% RSLogix 500 project WN16_175300_PPWEXT_04_2.rss, saved by version 9.00.00.04 %
PROJECT "EDIRX88"    % processor: SLC 500, 1747-L541 %

PROGRAM FILES
  LAD 2   13 rungs
  LAD 3   63 rungs
  LAD 4   5 rungs
  LAD 5   96 rungs
  LAD 6   14 rungs
  LAD 7   7 rungs
  LAD 8   17 rungs
  LAD 9   51 rungs
  LAD 10   4 rungs
  LAD 11   3 rungs
  LAD 12   6 rungs
  LAD 13   6 rungs
  LAD 14   6 rungs
  LAD 15   14 rungs
  LAD 16   7 rungs
  LAD 17   12 rungs
  LAD 18   4 rungs
  LAD 19   3 rungs
  LAD 21   27 rungs
  LAD 22   4 rungs
  LAD 23   7 rungs
  LAD 24   36 rungs

DATA FILES
  O0 OUTPUT  7 elements
  I1 INPUT  11 elements
  S2 STATUS  164 elements
  B3 BINARY  51 elements
  T4 TIMER  34 elements
  C5 COUNTER  1 elements
  R6 CONTROL  1 elements
  N7 INTEGER  241 elements
  F8 FLOAT  1 elements
  N9   24 elements
  N10   19 elements
  B13   10 elements
  T14   21 elements
  N17   100 elements
  N19   24 elements
  N20   11 elements
  N30   30 elements
  T31   10 elements

LADDER 2
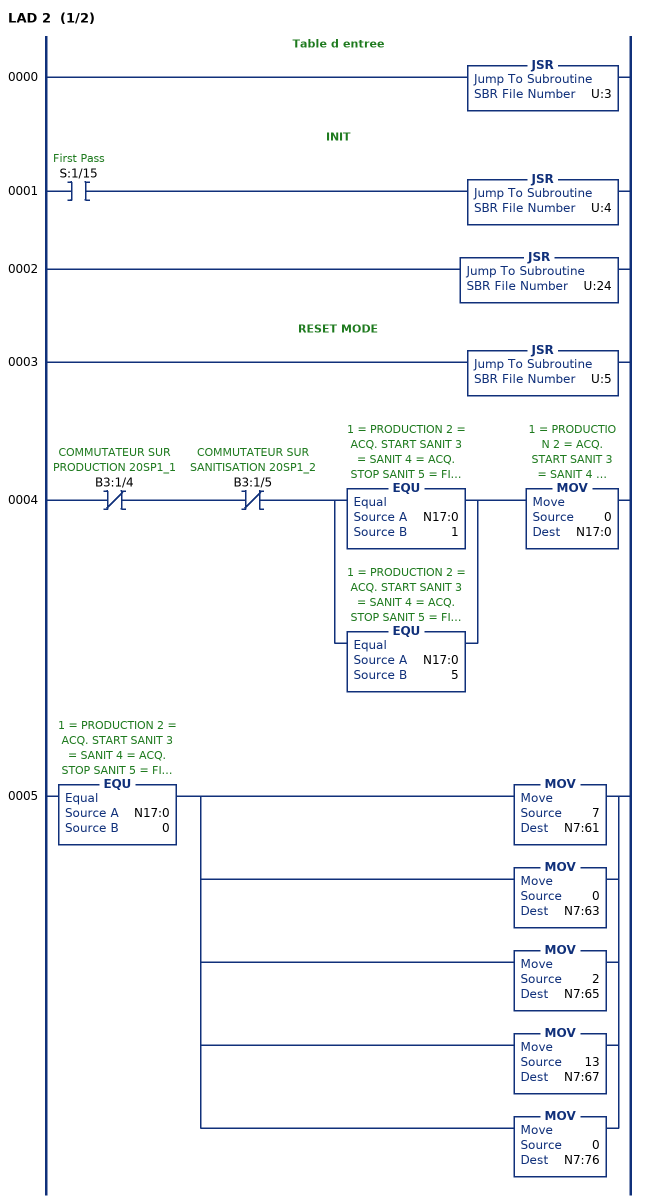
% Rung: 0 %
% TITLE: Table d entree %
SOR JSR U:3 EOR
% Rung: 1 %
% TITLE: INIT %
SOR XIC S:1/15 JSR U:4 EOR
%   S:1/15  "First Pass" %
% Rung: 2 %
SOR JSR U:24 EOR
% Rung: 3 %
% TITLE: RESET MODE %
SOR JSR U:5 EOR
% Rung: 4 %
SOR XIO B3:1/4 XIO B3:1/5 BST EQU N17:0 1 NXB EQU N17:0 5 BND MOV 0 N17:0 EOR
%   B3:1/4  20SP1_1  "COMMUTATEUR SUR PRODUCTION" %
%   B3:1/5  20SP1_2  "COMMUTATEUR SUR SANITISATION" %
%   N17:0  MODE  "1 = PRODUCTION 2 = ACQ. START SANIT 3 = SANIT 4 = ACQ. STOP SANIT 5 = FIN DE SANIT" %
% Rung: 5 %
SOR EQU N17:0 0 BST MOV 7 N7:61 NXB MOV 0 N7:63 NXB MOV 2 N7:65 NXB MOV 13 N7:67 NXB MOV 0 N7:76 BND EOR
%   N17:0  MODE  "1 = PRODUCTION 2 = ACQ. START SANIT 3 = SANIT 4 = ACQ. STOP SANIT 5 = FIN DE SANIT" %

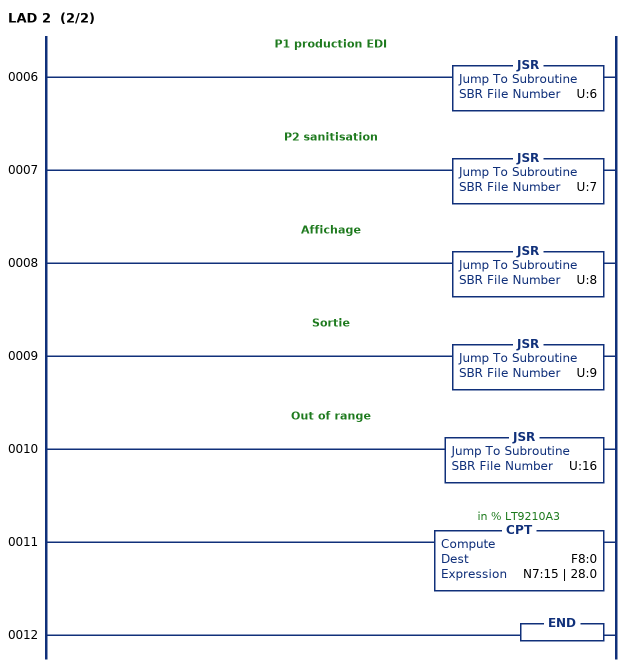
% Rung: 6 %
% TITLE: P1 production EDI %
SOR JSR U:6 EOR
% Rung: 7 %
% TITLE: P2 sanitisation %
SOR JSR U:7 EOR
% Rung: 8 %
% TITLE: Affichage %
SOR JSR U:8 EOR
% Rung: 9 %
% TITLE: Sortie %
SOR JSR U:9 EOR
% Rung: 10 %
% TITLE: Out of range %
SOR JSR U:16 EOR
% Rung: 11 %
SOR CPT F8:0 " N7:15 | 28.0 " EOR
%   F8:0  LT9210A3  "in %" %
%   N7:15  LT_VS_9210_A3 %
% Rung: 12 %
SOR END EOR

LADDER 3
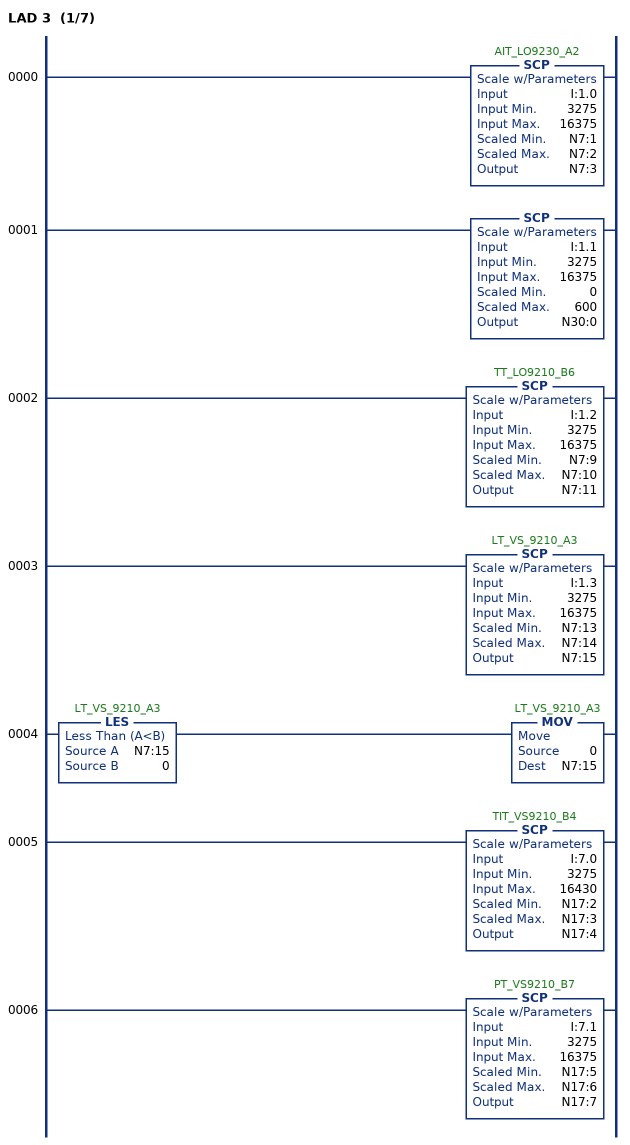
% Rung: 0 %
SOR SCP I:1.0 3275 16375 N7:1 N7:2 N7:3 EOR
%   N7:1  ZÉRO_AIT_LO9230_A2 %
%   N7:2  SPAN_AIT_LO9230_A2 %
%   N7:3  AIT_LO9230_A2 %
% Rung: 1 %
SOR SCP I:1.1 3275 16375 0 600 N30:0 EOR
% Rung: 2 %
SOR SCP I:1.2 3275 16375 N7:9 N7:10 N7:11 EOR
%   N7:9  ZÉRO_TT_LO9210_B6 %
%   N7:10  SPAN_TT_LO9210_B6 %
%   N7:11  TT_LO9210_B6 %
% Rung: 3 %
SOR SCP I:1.3 3275 16375 N7:13 N7:14 N7:15 EOR
%   N7:13  ZERO_LT_VS9210_A3 %
%   N7:14  SPAN_LT_VS9210_A3 %
%   N7:15  LT_VS_9210_A3 %
% Rung: 4 %
SOR LES N7:15 0 MOV 0 N7:15 EOR
%   N7:15  LT_VS_9210_A3 %
% Rung: 5 %
SOR SCP I:7.0 3275 16430 N17:2 N17:3 N17:4 EOR
%   N17:2  ZERO_TIT_VS9210_B4 %
%   N17:3  SPAN_TIT_VS9210_B4 %
%   N17:4  TIT_VS9210_B4 %
% Rung: 6 %
SOR SCP I:7.1 3275 16375 N17:5 N17:6 N17:7 EOR
%   N17:5  ZERO_PT_VS9210_B7 %
%   N17:6  SPAN_PT_VS9210_B7 %
%   N17:7  PT_VS9210_B7 %

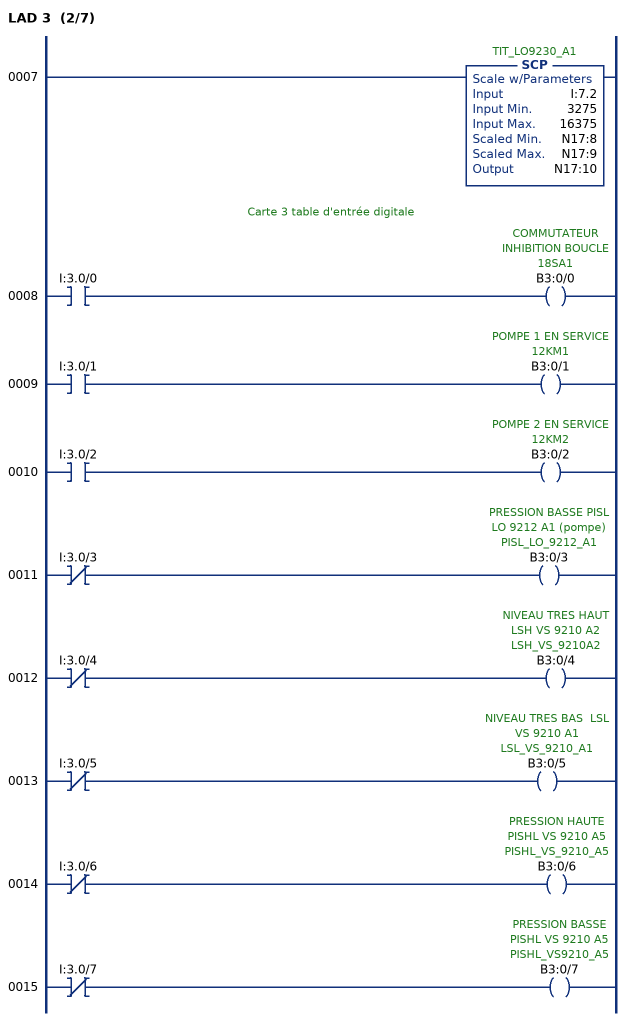
% Rung: 7 %
SOR SCP I:7.2 3275 16375 N17:8 N17:9 N17:10 EOR
%   N17:8  ZERO_TIT_LO9230_A1 %
%   N17:9  SPAN_TIT_LO9230_A1 %
%   N17:10  TIT_LO9230_A1 %
% Rung: 8 %
% Carte 3 table d'entrée digitale %
SOR XIC I:3.0/0 OTE B3:0/0 EOR
%   B3:0/0  18SA1  "COMMUTATEUR INHIBITION BOUCLE" %
% Rung: 9 %
SOR XIC I:3.0/1 OTE B3:0/1 EOR
%   B3:0/1  12KM1  "POMPE 1 EN SERVICE" %
% Rung: 10 %
SOR XIC I:3.0/2 OTE B3:0/2 EOR
%   B3:0/2  12KM2  "POMPE 2 EN SERVICE" %
% Rung: 11 %
SOR XIO I:3.0/3 OTE B3:0/3 EOR
%   B3:0/3  PISL_LO_9212_A1  "PRESSION BASSE PISL LO 9212 A1 (pompe)" %
% Rung: 12 %
SOR XIO I:3.0/4 OTE B3:0/4 EOR
%   B3:0/4  LSH_VS_9210A2  "NIVEAU TRES HAUT LSH VS 9210 A2" %
% Rung: 13 %
SOR XIO I:3.0/5 OTE B3:0/5 EOR
%   B3:0/5  LSL_VS_9210_A1  "NIVEAU TRES BAS  LSL VS 9210 A1" %
% Rung: 14 %
SOR XIO I:3.0/6 OTE B3:0/6 EOR
%   B3:0/6  PISHL_VS_9210_A5  "PRESSION HAUTE PISHL VS 9210 A5" %
% Rung: 15 %
SOR XIO I:3.0/7 OTE B3:0/7 EOR
%   B3:0/7  PISHL_VS9210_A5  "PRESSION BASSE PISHL VS 9210 A5" %

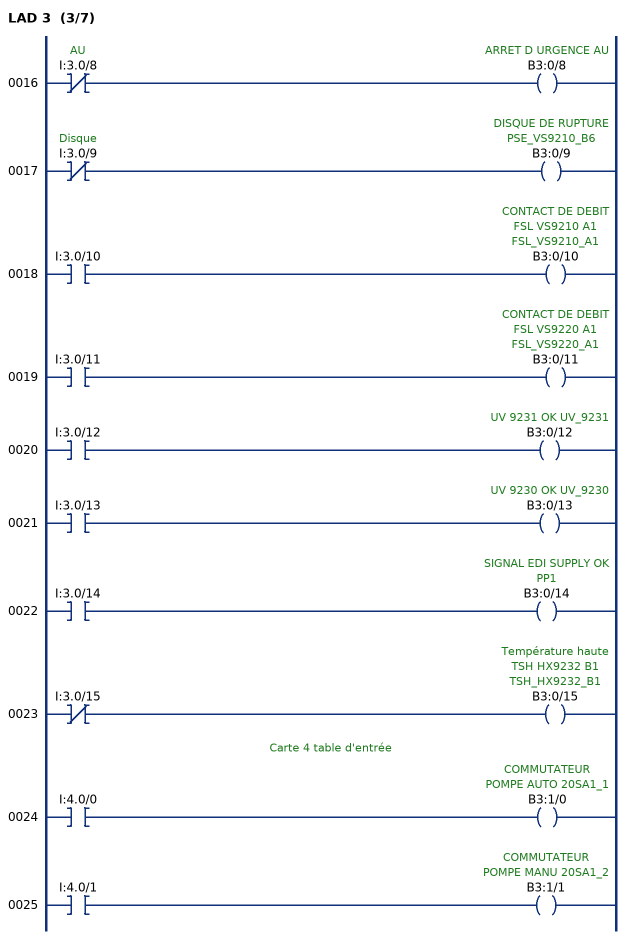
% Rung: 16 %
SOR XIO I:3.0/8 OTE B3:0/8 EOR
%   I:3.0/8  "AU" %
%   B3:0/8  AU  "ARRET D URGENCE" %
% Rung: 17 %
SOR XIO I:3.0/9 OTE B3:0/9 EOR
%   I:3.0/9  "Disque" %
%   B3:0/9  PSE_VS9210_B6  "DISQUE DE RUPTURE" %
% Rung: 18 %
SOR XIC I:3.0/10 OTE B3:0/10 EOR
%   B3:0/10  FSL_VS9210_A1  "CONTACT DE DEBIT FSL VS9210 A1" %
% Rung: 19 %
SOR XIC I:3.0/11 OTE B3:0/11 EOR
%   B3:0/11  FSL_VS9220_A1  "CONTACT DE DEBIT FSL VS9220 A1" %
% Rung: 20 %
SOR XIC I:3.0/12 OTE B3:0/12 EOR
%   B3:0/12  UV_9231  "UV 9231 OK" %
% Rung: 21 %
SOR XIC I:3.0/13 OTE B3:0/13 EOR
%   B3:0/13  UV_9230  "UV 9230 OK" %
% Rung: 22 %
SOR XIC I:3.0/14 OTE B3:0/14 EOR
%   B3:0/14  PP1  "SIGNAL EDI SUPPLY OK" %
% Rung: 23 %
SOR XIO I:3.0/15 OTE B3:0/15 EOR
%   B3:0/15  TSH_HX9232_B1  "Température haute TSH HX9232 B1" %
% Rung: 24 %
% Carte 4 table d'entrée %
SOR XIC I:4.0/0 OTE B3:1/0 EOR
%   B3:1/0  20SA1_1  "COMMUTATEUR POMPE AUTO" %
% Rung: 25 %
SOR XIC I:4.0/1 OTE B3:1/1 EOR
%   B3:1/1  20SA1_2  "COMMUTATEUR POMPE MANU" %

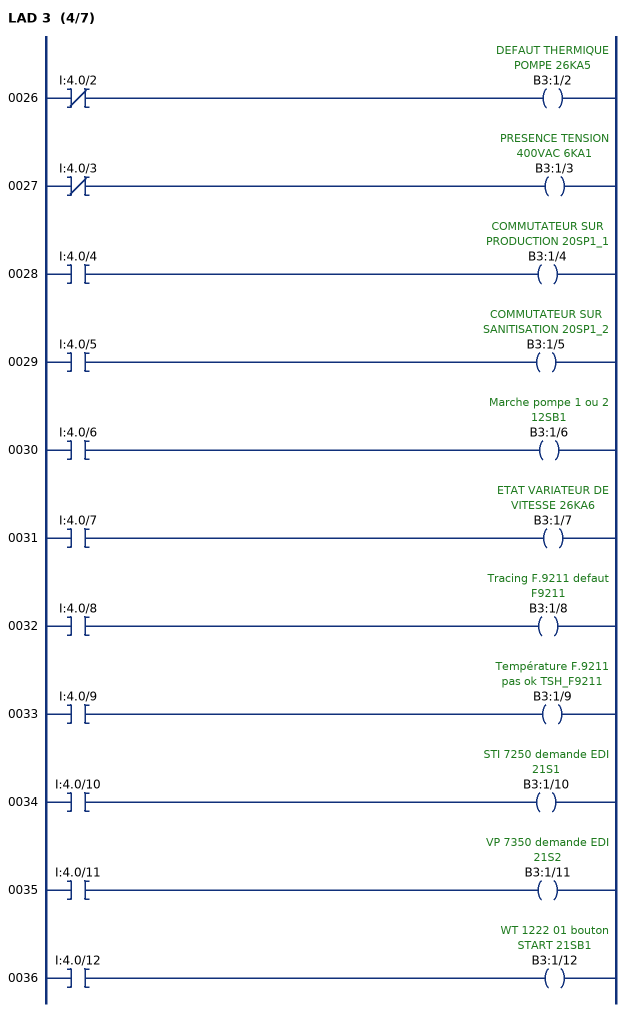
% Rung: 26 %
SOR XIO I:4.0/2 OTE B3:1/2 EOR
%   B3:1/2  26KA5  "DEFAUT THERMIQUE POMPE" %
% Rung: 27 %
SOR XIO I:4.0/3 OTE B3:1/3 EOR
%   B3:1/3  6KA1  "PRESENCE TENSION 400VAC" %
% Rung: 28 %
SOR XIC I:4.0/4 OTE B3:1/4 EOR
%   B3:1/4  20SP1_1  "COMMUTATEUR SUR PRODUCTION" %
% Rung: 29 %
SOR XIC I:4.0/5 OTE B3:1/5 EOR
%   B3:1/5  20SP1_2  "COMMUTATEUR SUR SANITISATION" %
% Rung: 30 %
SOR XIC I:4.0/6 OTE B3:1/6 EOR
%   B3:1/6  12SB1  "Marche pompe 1 ou 2" %
% Rung: 31 %
SOR XIC I:4.0/7 OTE B3:1/7 EOR
%   B3:1/7  26KA6  "ETAT VARIATEUR DE VITESSE" %
% Rung: 32 %
SOR XIC I:4.0/8 OTE B3:1/8 EOR
%   B3:1/8  F9211  "Tracing F.9211 defaut" %
% Rung: 33 %
SOR XIC I:4.0/9 OTE B3:1/9 EOR
%   B3:1/9  TSH_F9211  "Température F.9211 pas ok" %
% Rung: 34 %
SOR XIC I:4.0/10 OTE B3:1/10 EOR
%   B3:1/10  21S1  "STI 7250 demande EDI" %
% Rung: 35 %
SOR XIC I:4.0/11 OTE B3:1/11 EOR
%   B3:1/11  21S2  "VP 7350 demande EDI" %
% Rung: 36 %
SOR XIC I:4.0/12 OTE B3:1/12 EOR
%   B3:1/12  21SB1  "WT 1222 01 bouton START" %

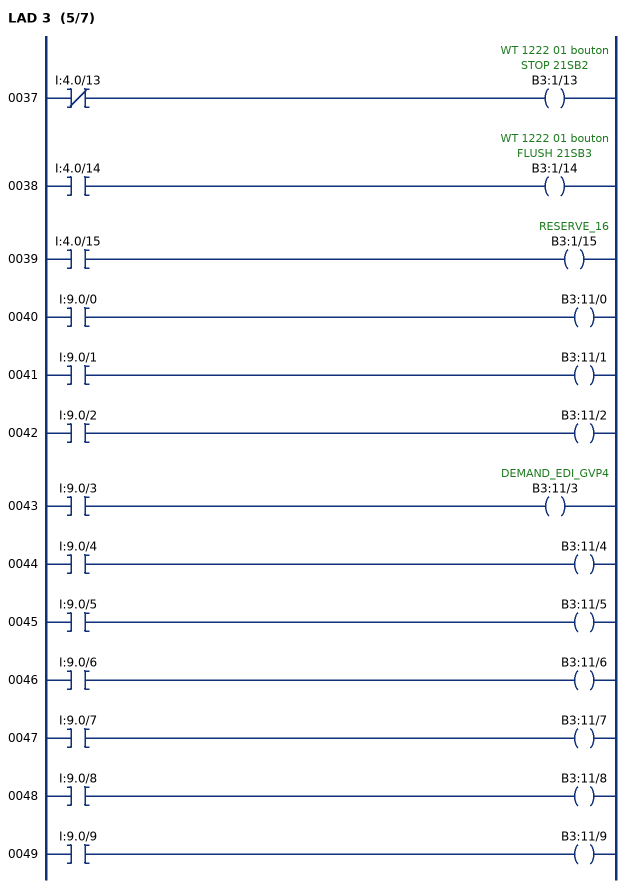
% Rung: 37 %
SOR XIO I:4.0/13 OTE B3:1/13 EOR
%   B3:1/13  21SB2  "WT 1222 01 bouton STOP" %
% Rung: 38 %
SOR XIC I:4.0/14 OTE B3:1/14 EOR
%   B3:1/14  21SB3  "WT 1222 01 bouton FLUSH" %
% Rung: 39 %
SOR XIC I:4.0/15 OTE B3:1/15 EOR
%   B3:1/15  RESERVE_16 %
% Rung: 40 %
SOR XIC I:9.0/0 OTE B3:11/0 EOR
% Rung: 41 %
SOR XIC I:9.0/1 OTE B3:11/1 EOR
% Rung: 42 %
SOR XIC I:9.0/2 OTE B3:11/2 EOR
% Rung: 43 %
SOR XIC I:9.0/3 OTE B3:11/3 EOR
%   B3:11/3  "DEMAND_EDI_GVP4" %
% Rung: 44 %
SOR XIC I:9.0/4 OTE B3:11/4 EOR
% Rung: 45 %
SOR XIC I:9.0/5 OTE B3:11/5 EOR
% Rung: 46 %
SOR XIC I:9.0/6 OTE B3:11/6 EOR
% Rung: 47 %
SOR XIC I:9.0/7 OTE B3:11/7 EOR
% Rung: 48 %
SOR XIC I:9.0/8 OTE B3:11/8 EOR
% Rung: 49 %
SOR XIC I:9.0/9 OTE B3:11/9 EOR

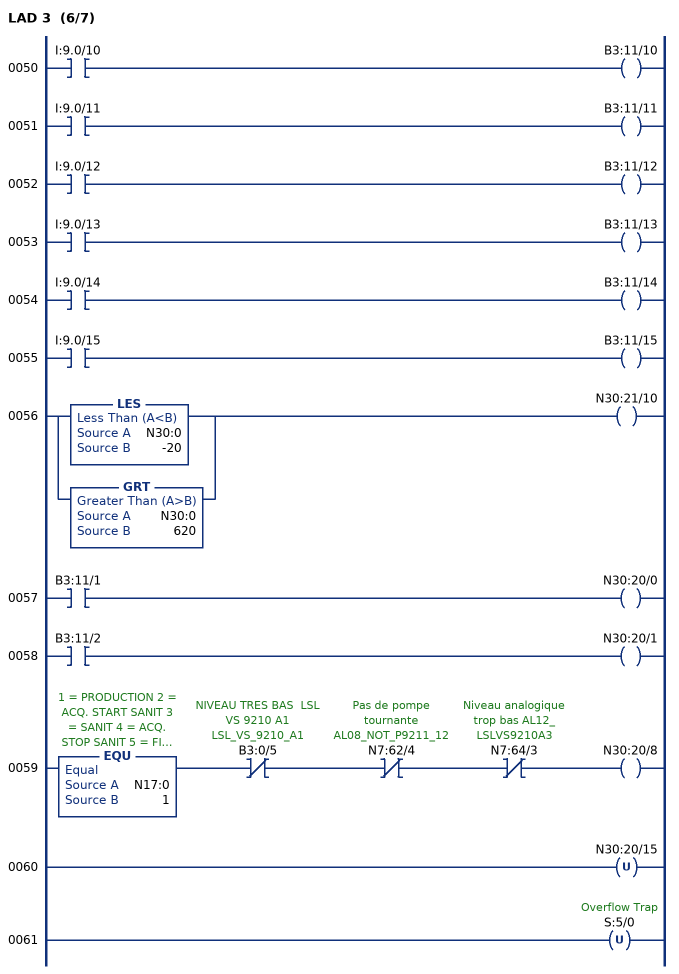
% Rung: 50 %
SOR XIC I:9.0/10 OTE B3:11/10 EOR
% Rung: 51 %
SOR XIC I:9.0/11 OTE B3:11/11 EOR
% Rung: 52 %
SOR XIC I:9.0/12 OTE B3:11/12 EOR
% Rung: 53 %
SOR XIC I:9.0/13 OTE B3:11/13 EOR
% Rung: 54 %
SOR XIC I:9.0/14 OTE B3:11/14 EOR
% Rung: 55 %
SOR XIC I:9.0/15 OTE B3:11/15 EOR
% Rung: 56 %
SOR BST LES N30:0 -20 NXB GRT N30:0 620 BND OTE N30:21/10 EOR
% Rung: 57 %
SOR XIC B3:11/1 OTE N30:20/0 EOR
% Rung: 58 %
SOR XIC B3:11/2 OTE N30:20/1 EOR
% Rung: 59 %
SOR EQU N17:0 1 XIO B3:0/5 XIO N7:62/4 XIO N7:64/3 OTE N30:20/8 EOR
%   N17:0  MODE  "1 = PRODUCTION 2 = ACQ. START SANIT 3 = SANIT 4 = ACQ. STOP SANIT 5 = FIN DE SANIT" %
%   B3:0/5  LSL_VS_9210_A1  "NIVEAU TRES BAS  LSL VS 9210 A1" %
%   N7:62/4  AL08_NOT_P9211_12  "Pas de pompe tournante" %
%   N7:64/3  AL12_LSLVS9210A3  "Niveau analogique trop bas" %
% Rung: 60 %
SOR OTU N30:20/15 EOR
% Rung: 61 %
SOR OTU S:5/0 EOR
%   S:5/0  "Overflow Trap" %

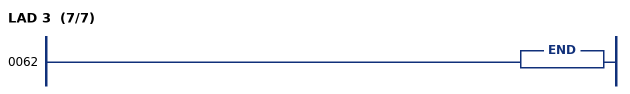
% Rung: 62 %
SOR END EOR

LADDER 4
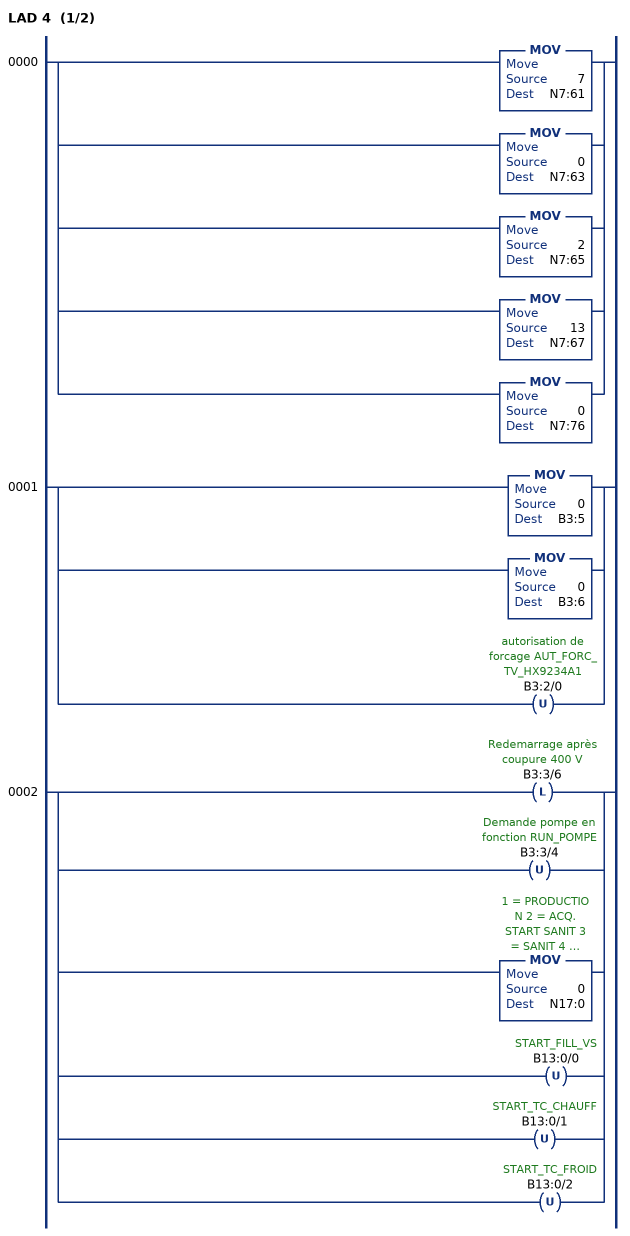
% Rung: 0 %
SOR BST MOV 7 N7:61 NXB MOV 0 N7:63 NXB MOV 2 N7:65 NXB MOV 13 N7:67 NXB MOV 0 N7:76 BND EOR
% Rung: 1 %
SOR BST MOV 0 B3:5 NXB MOV 0 B3:6 NXB OTU B3:2/0 BND EOR
%   B3:2/0  AUT_FORC_TV_HX9234A1  "autorisation de forcage" %
% Rung: 2 %
SOR BST OTL B3:3/6 NXB OTU B3:3/4 NXB MOV 0 N17:0 NXB OTU B13:0/0 NXB OTU B13:0/1 NXB OTU B13:0/2 BND EOR
%   B3:3/6  "Redemarrage après coupure 400 V" %
%   B3:3/4  RUN_POMPE  "Demande pompe en fonction" %
%   N17:0  MODE  "1 = PRODUCTION 2 = ACQ. START SANIT 3 = SANIT 4 = ACQ. STOP SANIT 5 = FIN DE SANIT" %
%   B13:0/0  START_FILL_VS %
%   B13:0/1  START_TC_CHAUFF %
%   B13:0/2  START_TC_FROID %

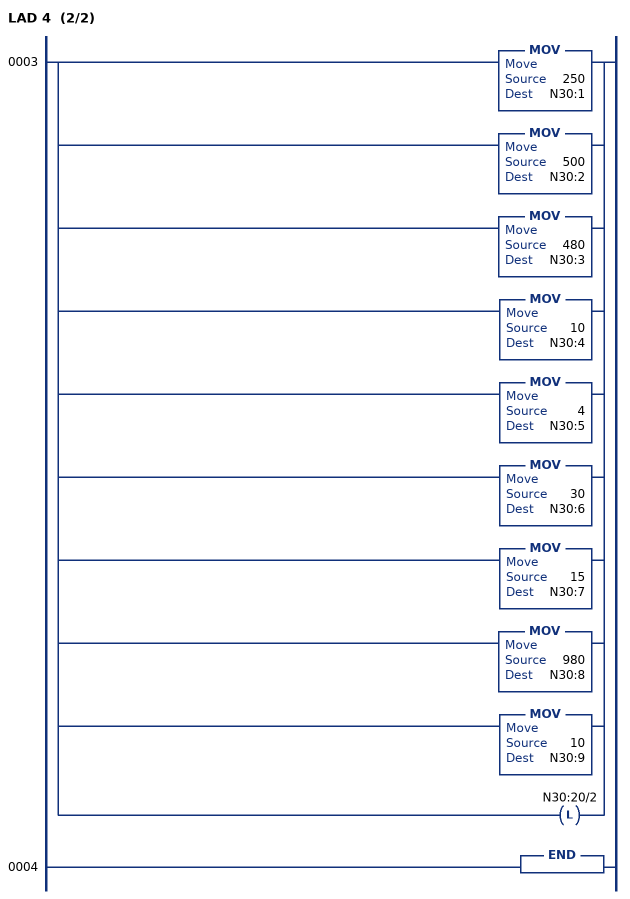
% Rung: 3 %
SOR BST MOV 250 N30:1 NXB MOV 500 N30:2 NXB MOV 480 N30:3 NXB MOV 10 N30:4 NXB MOV 4 N30:5 NXB MOV 30 N30:6 NXB MOV 15 N30:7 NXB MOV 980 N30:8 NXB MOV 10 N30:9 NXB OTL N30:20/2 BND EOR
% Rung: 4 %
SOR END EOR

LADDER 5
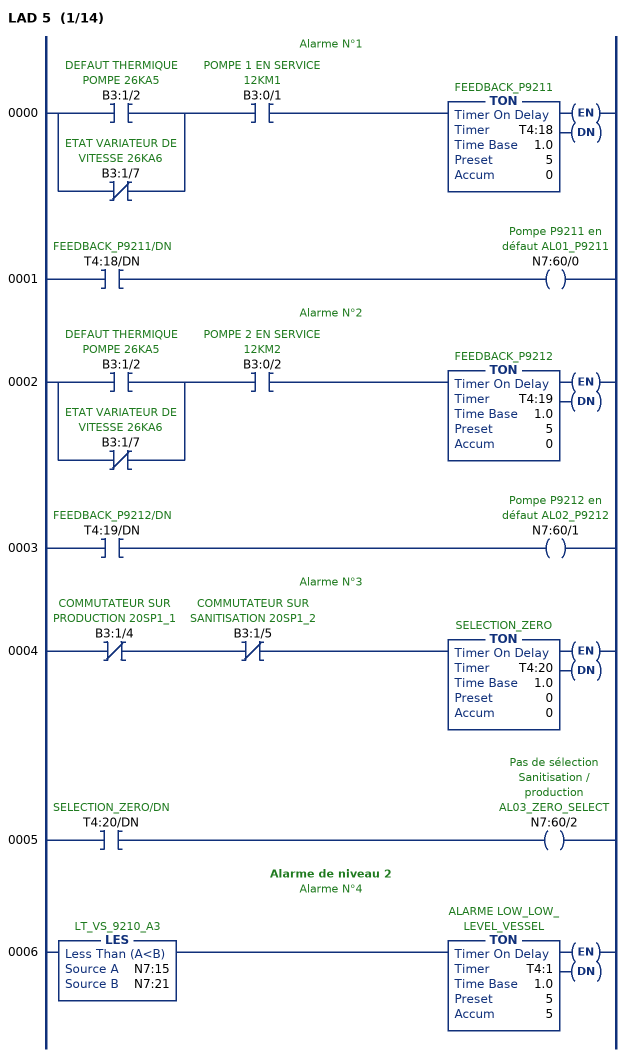
% Rung: 0 %
% Alarme N°1 %
SOR BST XIC B3:1/2 NXB XIO B3:1/7 BND XIC B3:0/1 TON T4:18 1.0 5 0 EOR
%   B3:1/2  26KA5  "DEFAUT THERMIQUE POMPE" %
%   B3:1/7  26KA6  "ETAT VARIATEUR DE VITESSE" %
%   B3:0/1  12KM1  "POMPE 1 EN SERVICE" %
%   T4:18  FEEDBACK_P9211 %
% Rung: 1 %
SOR XIC T4:18/DN OTE N7:60/0 EOR
%   T4:18  FEEDBACK_P9211 %
%   N7:60/0  AL01_P9211  "Pompe P9211 en défaut" %
% Rung: 2 %
% Alarme N°2 %
SOR BST XIC B3:1/2 NXB XIO B3:1/7 BND XIC B3:0/2 TON T4:19 1.0 5 0 EOR
%   B3:1/2  26KA5  "DEFAUT THERMIQUE POMPE" %
%   B3:1/7  26KA6  "ETAT VARIATEUR DE VITESSE" %
%   B3:0/2  12KM2  "POMPE 2 EN SERVICE" %
%   T4:19  FEEDBACK_P9212 %
% Rung: 3 %
SOR XIC T4:19/DN OTE N7:60/1 EOR
%   T4:19  FEEDBACK_P9212 %
%   N7:60/1  AL02_P9212  "Pompe P9212 en défaut" %
% Rung: 4 %
% Alarme N°3 %
SOR XIO B3:1/4 XIO B3:1/5 TON T4:20 1.0 0 0 EOR
%   B3:1/4  20SP1_1  "COMMUTATEUR SUR PRODUCTION" %
%   B3:1/5  20SP1_2  "COMMUTATEUR SUR SANITISATION" %
%   T4:20  SELECTION_ZERO %
% Rung: 5 %
SOR XIC T4:20/DN OTE N7:60/2 EOR
%   T4:20  SELECTION_ZERO %
%   N7:60/2  AL03_ZERO_SELECT  "Pas de sélection Sanitisation / production" %
% Rung: 6 %
% TITLE: Alarme de niveau 2 %
% Alarme N°4 %
SOR LES N7:15 N7:21 TON T4:1 1.0 5 5 EOR
%   N7:15  LT_VS_9210_A3 %
%   N7:21  LSLL_9210_A3 %
%   T4:1  LOW_LOW_LEVEL_VESSEL  "ALARME" %

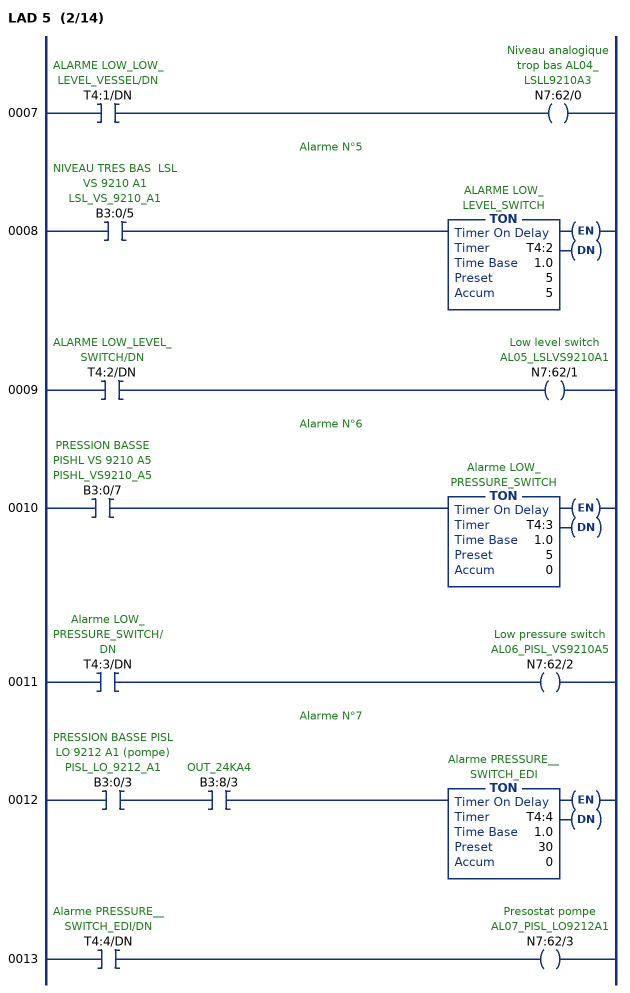
% Rung: 7 %
SOR XIC T4:1/DN OTE N7:62/0 EOR
%   T4:1  LOW_LOW_LEVEL_VESSEL  "ALARME" %
%   N7:62/0  AL04_LSLL9210A3  "Niveau analogique trop bas" %
% Rung: 8 %
% Alarme N°5 %
SOR XIC B3:0/5 TON T4:2 1.0 5 5 EOR
%   B3:0/5  LSL_VS_9210_A1  "NIVEAU TRES BAS  LSL VS 9210 A1" %
%   T4:2  LOW_LEVEL_SWITCH  "ALARME" %
% Rung: 9 %
SOR XIC T4:2/DN OTE N7:62/1 EOR
%   T4:2  LOW_LEVEL_SWITCH  "ALARME" %
%   N7:62/1  AL05_LSLVS9210A1  "Low level switch" %
% Rung: 10 %
% Alarme N°6 %
SOR XIC B3:0/7 TON T4:3 1.0 5 0 EOR
%   B3:0/7  PISHL_VS9210_A5  "PRESSION BASSE PISHL VS 9210 A5" %
%   T4:3  LOW_PRESSURE_SWITCH  "Alarme" %
% Rung: 11 %
SOR XIC T4:3/DN OTE N7:62/2 EOR
%   T4:3  LOW_PRESSURE_SWITCH  "Alarme" %
%   N7:62/2  AL06_PISL_VS9210A5  "Low pressure switch" %
% Rung: 12 %
% Alarme N°7 %
SOR XIC B3:0/3 XIC B3:8/3 TON T4:4 1.0 30 0 EOR
%   B3:0/3  PISL_LO_9212_A1  "PRESSION BASSE PISL LO 9212 A1 (pompe)" %
%   B3:8/3  "OUT_24KA4" %
%   T4:4  PRESSURE__SWITCH_EDI  "Alarme" %
% Rung: 13 %
SOR XIC T4:4/DN OTE N7:62/3 EOR
%   T4:4  PRESSURE__SWITCH_EDI  "Alarme" %
%   N7:62/3  AL07_PISL_LO9212A1  "Presostat pompe" %

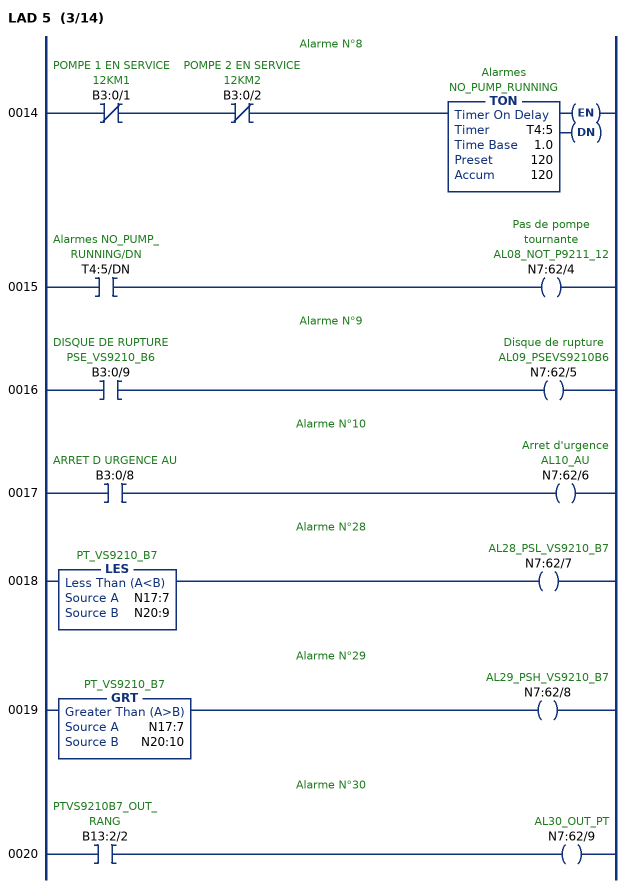
% Rung: 14 %
% Alarme N°8 %
SOR XIO B3:0/1 XIO B3:0/2 TON T4:5 1.0 120 120 EOR
%   B3:0/1  12KM1  "POMPE 1 EN SERVICE" %
%   B3:0/2  12KM2  "POMPE 2 EN SERVICE" %
%   T4:5  NO_PUMP_RUNNING  "Alarmes" %
% Rung: 15 %
SOR XIC T4:5/DN OTE N7:62/4 EOR
%   T4:5  NO_PUMP_RUNNING  "Alarmes" %
%   N7:62/4  AL08_NOT_P9211_12  "Pas de pompe tournante" %
% Rung: 16 %
% Alarme N°9 %
SOR XIC B3:0/9 OTE N7:62/5 EOR
%   B3:0/9  PSE_VS9210_B6  "DISQUE DE RUPTURE" %
%   N7:62/5  AL09_PSEVS9210B6  "Disque de rupture" %
% Rung: 17 %
% Alarme N°10 %
SOR XIC B3:0/8 OTE N7:62/6 EOR
%   B3:0/8  AU  "ARRET D URGENCE" %
%   N7:62/6  AL10_AU  "Arret d'urgence" %
% Rung: 18 %
% Alarme N°28 %
SOR LES N17:7 N20:9 OTE N7:62/7 EOR
%   N17:7  PT_VS9210_B7 %
%   N20:9  PSL_VS9210_B7 %
%   N7:62/7  AL28_PSL_VS9210_B7 %
% Rung: 19 %
% Alarme N°29 %
SOR GRT N17:7 N20:10 OTE N7:62/8 EOR
%   N17:7  PT_VS9210_B7 %
%   N20:10  PSH_VS9210_B7 %
%   N7:62/8  AL29_PSH_VS9210_B7 %
% Rung: 20 %
% Alarme N°30 %
SOR XIC B13:2/2 OTE N7:62/9 EOR
%   B13:2/2  PTVS9210B7_OUT_RANG %
%   N7:62/9  AL30_OUT_PT %

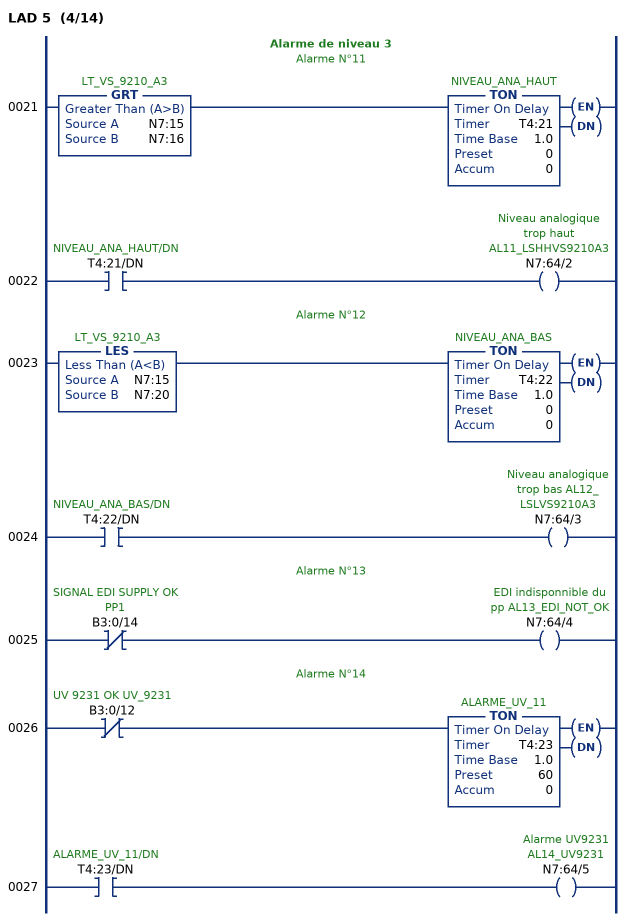
% Rung: 21 %
% TITLE: Alarme de niveau 3 %
% Alarme N°11 %
SOR GRT N7:15 N7:16 TON T4:21 1.0 0 0 EOR
%   N7:15  LT_VS_9210_A3 %
%   N7:16  LSHH_VS9210_A3 %
%   T4:21  NIVEAU_ANA_HAUT %
% Rung: 22 %
SOR XIC T4:21/DN OTE N7:64/2 EOR
%   T4:21  NIVEAU_ANA_HAUT %
%   N7:64/2  AL11_LSHHVS9210A3  "Niveau analogique trop haut" %
% Rung: 23 %
% Alarme N°12 %
SOR LES N7:15 N7:20 TON T4:22 1.0 0 0 EOR
%   N7:15  LT_VS_9210_A3 %
%   N7:20  LSL_VS_9210_A3 %
%   T4:22  NIVEAU_ANA_BAS %
% Rung: 24 %
SOR XIC T4:22/DN OTE N7:64/3 EOR
%   T4:22  NIVEAU_ANA_BAS %
%   N7:64/3  AL12_LSLVS9210A3  "Niveau analogique trop bas" %
% Rung: 25 %
% Alarme N°13 %
SOR XIO B3:0/14 OTE N7:64/4 EOR
%   B3:0/14  PP1  "SIGNAL EDI SUPPLY OK" %
%   N7:64/4  AL13_EDI_NOT_OK  "EDI indisponnible du pp" %
% Rung: 26 %
% Alarme N°14 %
SOR XIO B3:0/12 TON T4:23 1.0 60 0 EOR
%   B3:0/12  UV_9231  "UV 9231 OK" %
%   T4:23  ALARME_UV_11 %
% Rung: 27 %
SOR XIC T4:23/DN OTE N7:64/5 EOR
%   T4:23  ALARME_UV_11 %
%   N7:64/5  AL14_UV9231  "Alarme UV9231" %

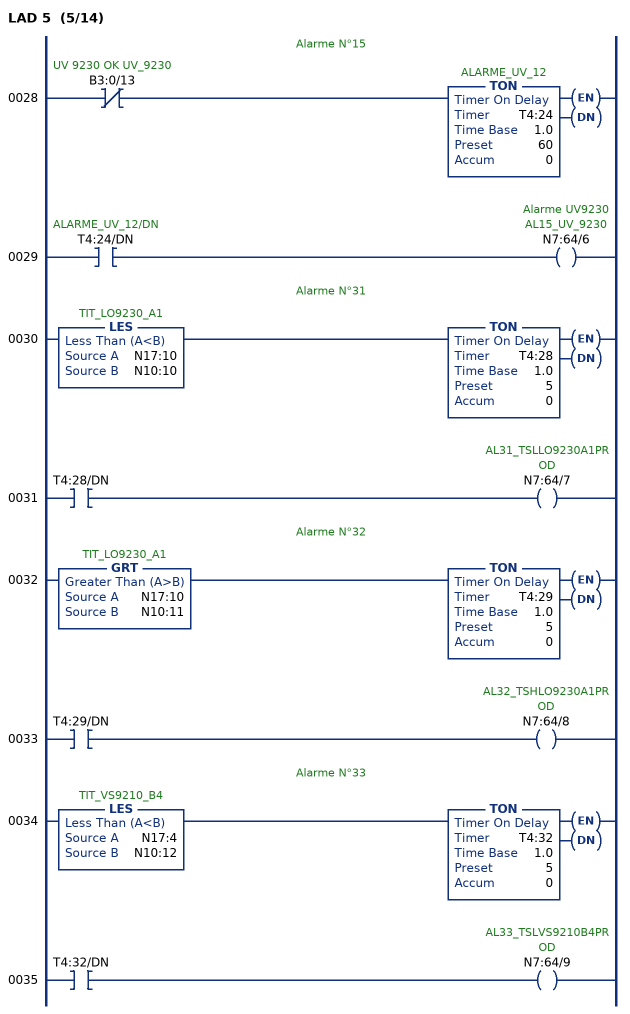
% Rung: 28 %
% Alarme N°15 %
SOR XIO B3:0/13 TON T4:24 1.0 60 0 EOR
%   B3:0/13  UV_9230  "UV 9230 OK" %
%   T4:24  ALARME_UV_12 %
% Rung: 29 %
SOR XIC T4:24/DN OTE N7:64/6 EOR
%   T4:24  ALARME_UV_12 %
%   N7:64/6  AL15_UV_9230  "Alarme UV9230" %
% Rung: 30 %
% Alarme N°31 %
SOR LES N17:10 N10:10 TON T4:28 1.0 5 0 EOR
%   N17:10  TIT_LO9230_A1 %
%   N10:10  TSLLO9230A1_PROD %
% Rung: 31 %
SOR XIC T4:28/DN OTE N7:64/7 EOR
%   N7:64/7  AL31_TSLLO9230A1PROD %
% Rung: 32 %
% Alarme N°32 %
SOR GRT N17:10 N10:11 TON T4:29 1.0 5 0 EOR
%   N17:10  TIT_LO9230_A1 %
%   N10:11  TSHLO9230A1_PROD %
% Rung: 33 %
SOR XIC T4:29/DN OTE N7:64/8 EOR
%   N7:64/8  AL32_TSHLO9230A1PROD %
% Rung: 34 %
% Alarme N°33 %
SOR LES N17:4 N10:12 TON T4:32 1.0 5 0 EOR
%   N17:4  TIT_VS9210_B4 %
%   N10:12  TSL_VS9210_B4_PROD %
% Rung: 35 %
SOR XIC T4:32/DN OTE N7:64/9 EOR
%   N7:64/9  AL33_TSLVS9210B4PROD %

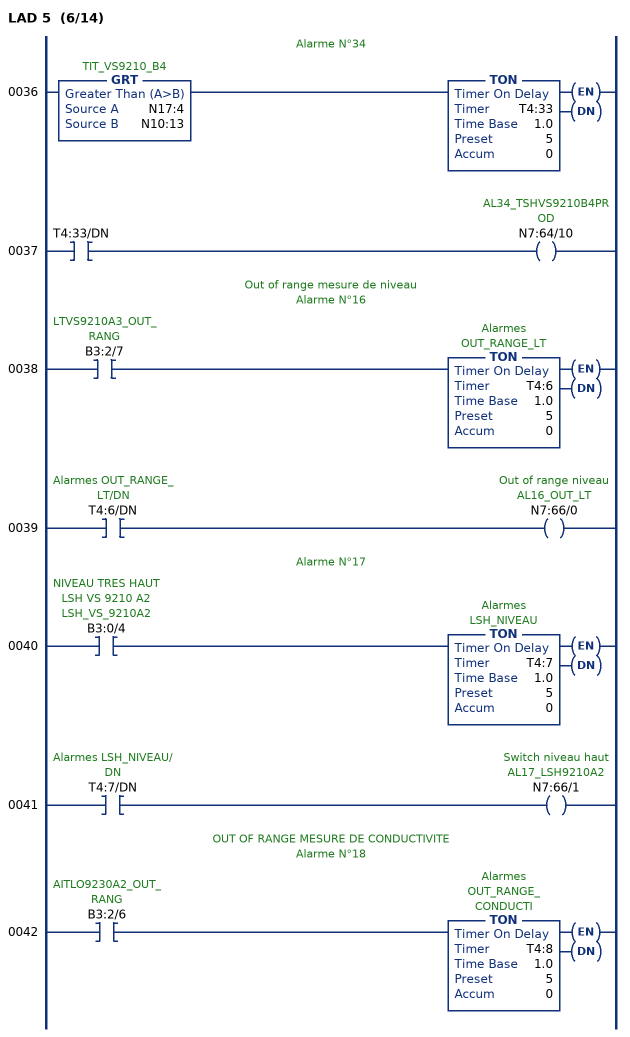
% Rung: 36 %
% Alarme N°34 %
SOR GRT N17:4 N10:13 TON T4:33 1.0 5 0 EOR
%   N17:4  TIT_VS9210_B4 %
%   N10:13  TSH_VS9210_B4_PROD %
% Rung: 37 %
SOR XIC T4:33/DN OTE N7:64/10 EOR
%   N7:64/10  AL34_TSHVS9210B4PROD %
% Rung: 38 %
% Out of range mesure de niveau
% Alarme N°16 %
SOR XIC B3:2/7 TON T4:6 1.0 5 0 EOR
%   B3:2/7  LTVS9210A3_OUT_RANG %
%   T4:6  OUT_RANGE_LT  "Alarmes" %
% Rung: 39 %
SOR XIC T4:6/DN OTE N7:66/0 EOR
%   T4:6  OUT_RANGE_LT  "Alarmes" %
%   N7:66/0  AL16_OUT_LT  "Out of range niveau" %
% Rung: 40 %
% Alarme N°17 %
SOR XIC B3:0/4 TON T4:7 1.0 5 0 EOR
%   B3:0/4  LSH_VS_9210A2  "NIVEAU TRES HAUT LSH VS 9210 A2" %
%   T4:7  LSH_NIVEAU  "Alarmes" %
% Rung: 41 %
SOR XIC T4:7/DN OTE N7:66/1 EOR
%   T4:7  LSH_NIVEAU  "Alarmes" %
%   N7:66/1  AL17_LSH9210A2  "Switch niveau haut" %
% Rung: 42 %
% OUT OF RANGE MESURE DE CONDUCTIVITE
% Alarme N°18 %
SOR XIC B3:2/6 TON T4:8 1.0 5 0 EOR
%   B3:2/6  AITLO9230A2_OUT_RANG %
%   T4:8  OUT_RANGE_CONDUCTI  "Alarmes" %

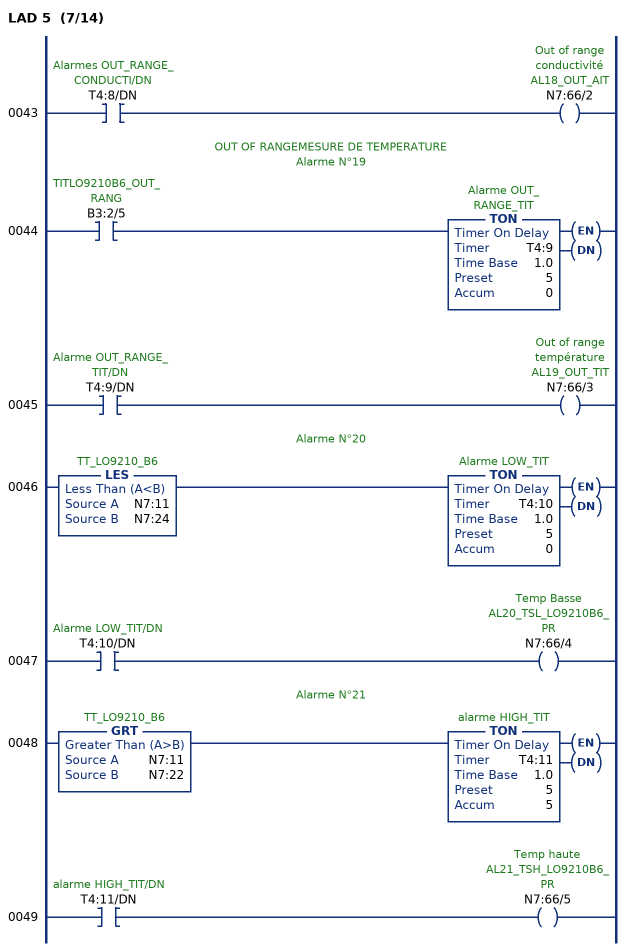
% Rung: 43 %
SOR XIC T4:8/DN OTE N7:66/2 EOR
%   T4:8  OUT_RANGE_CONDUCTI  "Alarmes" %
%   N7:66/2  AL18_OUT_AIT  "Out of range conductivité" %
% Rung: 44 %
% OUT OF RANGEMESURE DE TEMPERATURE
% Alarme N°19 %
SOR XIC B3:2/5 TON T4:9 1.0 5 0 EOR
%   B3:2/5  TITLO9210B6_OUT_RANG %
%   T4:9  OUT_RANGE_TIT  "Alarme" %
% Rung: 45 %
SOR XIC T4:9/DN OTE N7:66/3 EOR
%   T4:9  OUT_RANGE_TIT  "Alarme" %
%   N7:66/3  AL19_OUT_TIT  "Out of range température" %
% Rung: 46 %
% Alarme N°20 %
SOR LES N7:11 N7:24 TON T4:10 1.0 5 0 EOR
%   N7:11  TT_LO9210_B6 %
%   N7:24  TSL_LO9210B6  "TEMPERATURE DE RETOUR BOUCLE TROP BASSE" %
%   T4:10  LOW_TIT  "Alarme" %
% Rung: 47 %
SOR XIC T4:10/DN OTE N7:66/4 EOR
%   T4:10  LOW_TIT  "Alarme" %
%   N7:66/4  AL20_TSL_LO9210B6_PR  "Temp Basse" %
% Rung: 48 %
% Alarme N°21 %
SOR GRT N7:11 N7:22 TON T4:11 1.0 5 5 EOR
%   N7:11  TT_LO9210_B6 %
%   N7:22  TSH_LO9210B6_PR  "TEMPERATURE HAUTE RETOUR BOUCLE" %
%   T4:11  HIGH_TIT  "alarme" %
% Rung: 49 %
SOR XIC T4:11/DN OTE N7:66/5 EOR
%   T4:11  HIGH_TIT  "alarme" %
%   N7:66/5  AL21_TSH_LO9210B6_PR  "Temp haute" %

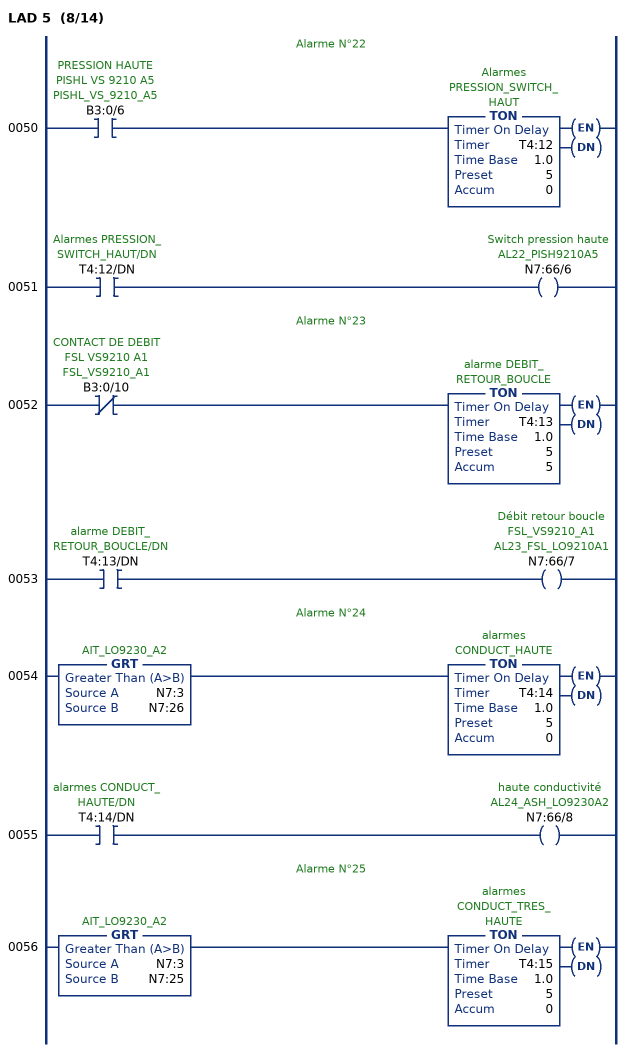
% Rung: 50 %
% Alarme N°22 %
SOR XIC B3:0/6 TON T4:12 1.0 5 0 EOR
%   B3:0/6  PISHL_VS_9210_A5  "PRESSION HAUTE PISHL VS 9210 A5" %
%   T4:12  PRESSION_SWITCH_HAUT  "Alarmes" %
% Rung: 51 %
SOR XIC T4:12/DN OTE N7:66/6 EOR
%   T4:12  PRESSION_SWITCH_HAUT  "Alarmes" %
%   N7:66/6  AL22_PISH9210A5  "Switch pression haute" %
% Rung: 52 %
% Alarme N°23 %
SOR XIO B3:0/10 TON T4:13 1.0 5 5 EOR
%   B3:0/10  FSL_VS9210_A1  "CONTACT DE DEBIT FSL VS9210 A1" %
%   T4:13  DEBIT_RETOUR_BOUCLE  "alarme" %
% Rung: 53 %
SOR XIC T4:13/DN OTE N7:66/7 EOR
%   T4:13  DEBIT_RETOUR_BOUCLE  "alarme" %
%   N7:66/7  AL23_FSL_LO9210A1  "Débit retour boucle FSL_VS9210_A1" %
% Rung: 54 %
% Alarme N°24 %
SOR GRT N7:3 N7:26 TON T4:14 1.0 5 0 EOR
%   N7:3  AIT_LO9230_A2 %
%   N7:26  ASH_LO_9230A2  "HIGH CONDUCTIVITY RETURN" %
%   T4:14  CONDUCT_HAUTE  "alarmes" %
% Rung: 55 %
SOR XIC T4:14/DN OTE N7:66/8 EOR
%   T4:14  CONDUCT_HAUTE  "alarmes" %
%   N7:66/8  AL24_ASH_LO9230A2  "haute conductivité" %
% Rung: 56 %
% Alarme N°25 %
SOR GRT N7:3 N7:25 TON T4:15 1.0 5 0 EOR
%   N7:3  AIT_LO9230_A2 %
%   N7:25  ASHH_LO9230A2  "HIGH HIGH CONDUCTIVITE RETURN" %
%   T4:15  CONDUCT_TRES_HAUTE  "alarmes" %

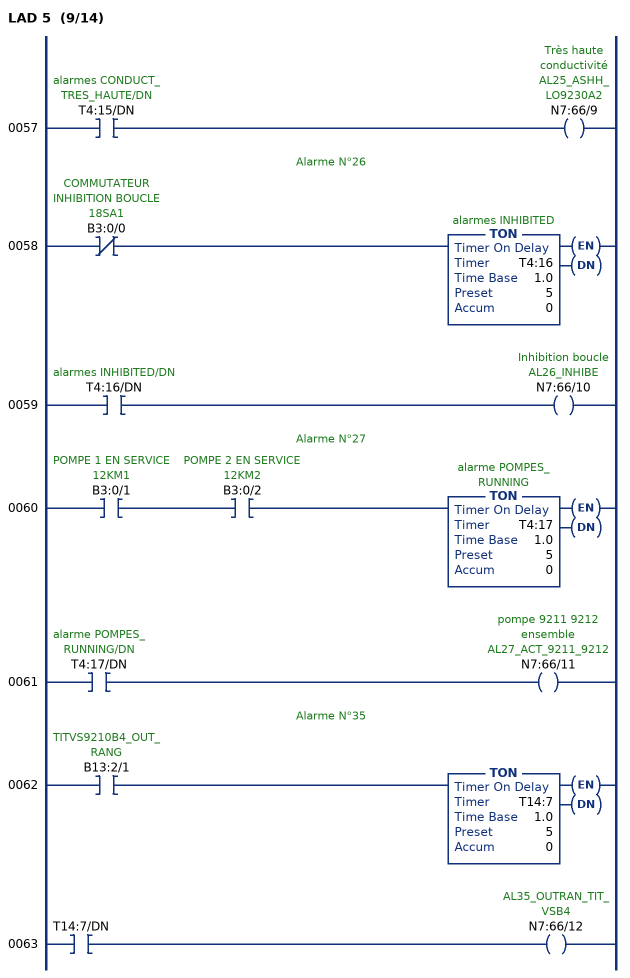
% Rung: 57 %
SOR XIC T4:15/DN OTE N7:66/9 EOR
%   T4:15  CONDUCT_TRES_HAUTE  "alarmes" %
%   N7:66/9  AL25_ASHH_LO9230A2  "Très haute conductivité" %
% Rung: 58 %
% Alarme N°26 %
SOR XIO B3:0/0 TON T4:16 1.0 5 0 EOR
%   B3:0/0  18SA1  "COMMUTATEUR INHIBITION BOUCLE" %
%   T4:16  INHIBITED  "alarmes" %
% Rung: 59 %
SOR XIC T4:16/DN OTE N7:66/10 EOR
%   T4:16  INHIBITED  "alarmes" %
%   N7:66/10  AL26_INHIBE  "Inhibition boucle" %
% Rung: 60 %
% Alarme N°27 %
SOR XIC B3:0/1 XIC B3:0/2 TON T4:17 1.0 5 0 EOR
%   B3:0/1  12KM1  "POMPE 1 EN SERVICE" %
%   B3:0/2  12KM2  "POMPE 2 EN SERVICE" %
%   T4:17  POMPES_RUNNING  "alarme" %
% Rung: 61 %
SOR XIC T4:17/DN OTE N7:66/11 EOR
%   T4:17  POMPES_RUNNING  "alarme" %
%   N7:66/11  AL27_ACT_9211_9212  "pompe 9211 9212 ensemble" %
% Rung: 62 %
% Alarme N°35 %
SOR XIC B13:2/1 TON T14:7 1.0 5 0 EOR
%   B13:2/1  TITVS9210B4_OUT_RANG %
% Rung: 63 %
SOR XIC T14:7/DN OTE N7:66/12 EOR
%   N7:66/12  AL35_OUTRAN_TIT_VSB4 %

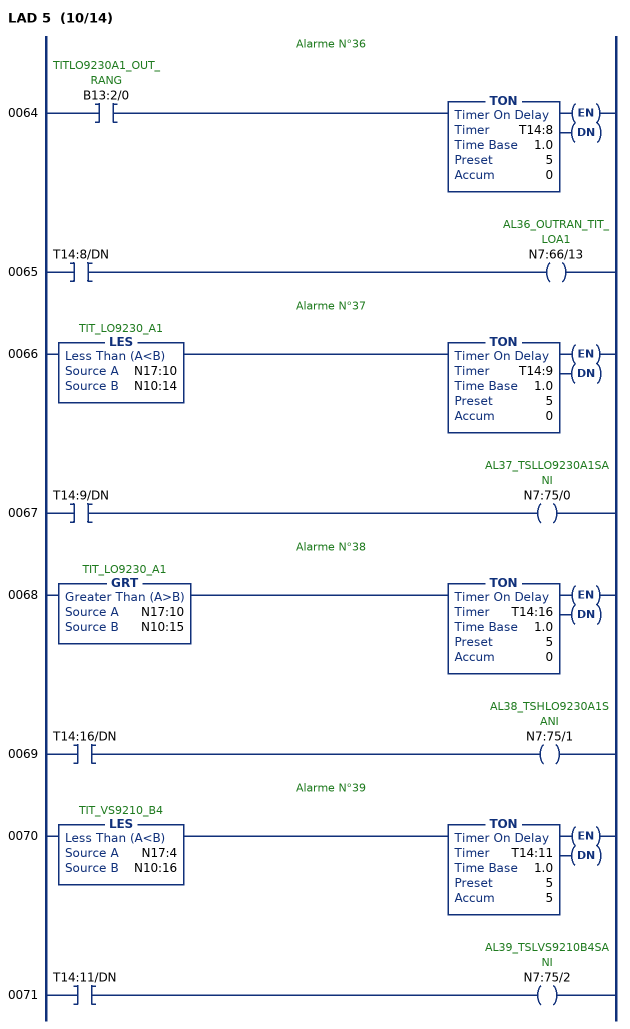
% Rung: 64 %
% Alarme N°36 %
SOR XIC B13:2/0 TON T14:8 1.0 5 0 EOR
%   B13:2/0  TITLO9230A1_OUT_RANG %
% Rung: 65 %
SOR XIC T14:8/DN OTE N7:66/13 EOR
%   N7:66/13  AL36_OUTRAN_TIT_LOA1 %
% Rung: 66 %
% Alarme N°37 %
SOR LES N17:10 N10:14 TON T14:9 1.0 5 0 EOR
%   N17:10  TIT_LO9230_A1 %
%   N10:14  TSL_LO9230_A1 %
% Rung: 67 %
SOR XIC T14:9/DN OTE N7:75/0 EOR
%   N7:75/0  AL37_TSLLO9230A1SANI %
% Rung: 68 %
% Alarme N°38 %
SOR GRT N17:10 N10:15 TON T14:16 1.0 5 0 EOR
%   N17:10  TIT_LO9230_A1 %
%   N10:15  TSH_LO9230_A1 %
% Rung: 69 %
SOR XIC T14:16/DN OTE N7:75/1 EOR
%   N7:75/1  AL38_TSHLO9230A1SANI %
% Rung: 70 %
% Alarme N°39 %
SOR LES N17:4 N10:16 TON T14:11 1.0 5 5 EOR
%   N17:4  TIT_VS9210_B4 %
%   N10:16  TSL_VS9210_B4_SANI %
% Rung: 71 %
SOR XIC T14:11/DN OTE N7:75/2 EOR
%   N7:75/2  AL39_TSLVS9210B4SANI %

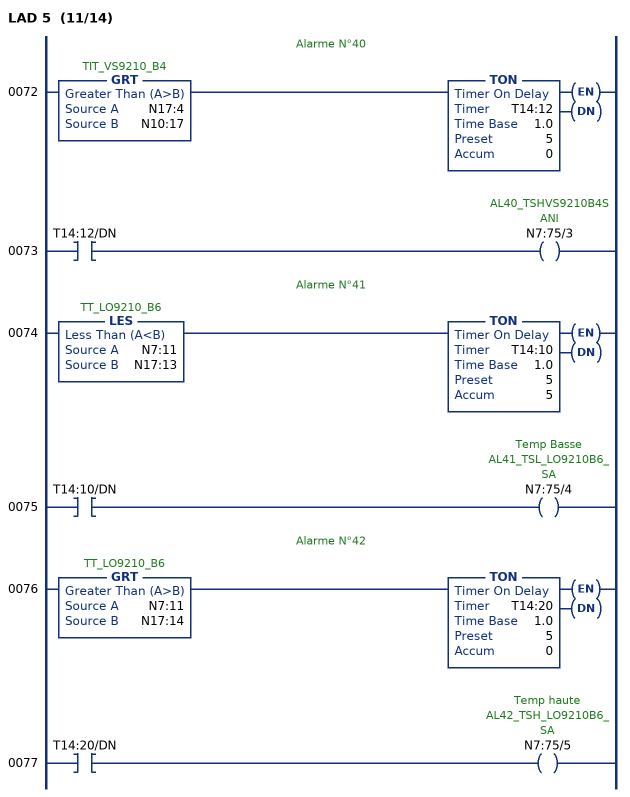
% Rung: 72 %
% Alarme N°40 %
SOR GRT N17:4 N10:17 TON T14:12 1.0 5 0 EOR
%   N17:4  TIT_VS9210_B4 %
%   N10:17  TSH_VS9210_B4_SANI %
% Rung: 73 %
SOR XIC T14:12/DN OTE N7:75/3 EOR
%   N7:75/3  AL40_TSHVS9210B4SANI %
% Rung: 74 %
% Alarme N°41 %
SOR LES N7:11 N17:13 TON T14:10 1.0 5 5 EOR
%   N7:11  TT_LO9210_B6 %
%   N17:13  TSL_LO9210B6_SANIT %
% Rung: 75 %
SOR XIC T14:10/DN OTE N7:75/4 EOR
%   N7:75/4  AL41_TSL_LO9210B6_SA  "Temp Basse" %
% Rung: 76 %
% Alarme N°42 %
SOR GRT N7:11 N17:14 TON T14:20 1.0 5 0 EOR
%   N7:11  TT_LO9210_B6 %
%   N17:14  TSH_LO9210B6_SANIT %
% Rung: 77 %
SOR XIC T14:20/DN OTE N7:75/5 EOR
%   N7:75/5  AL42_TSH_LO9210B6_SA  "Temp haute" %

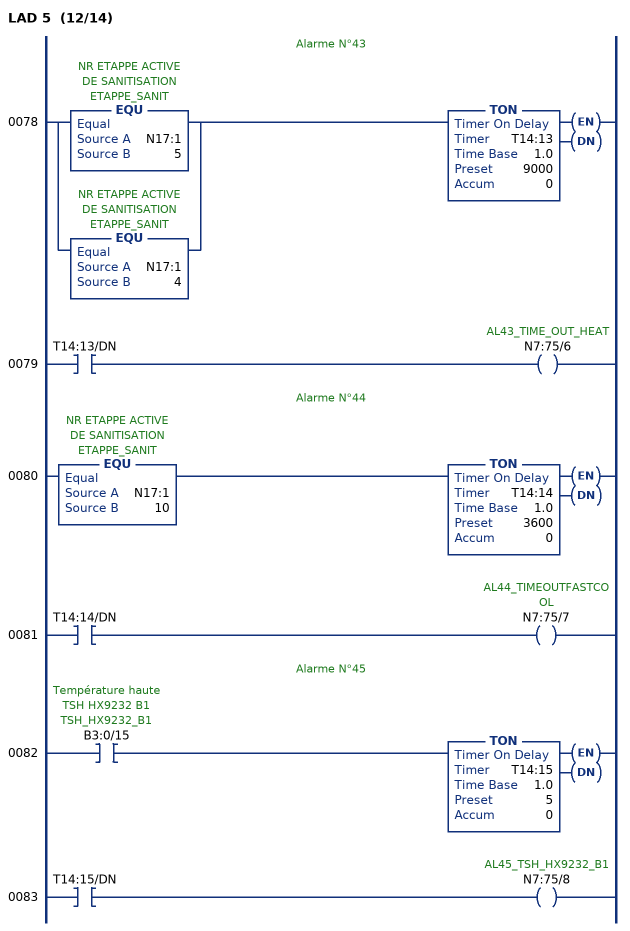
% Rung: 78 %
% Alarme N°43 %
SOR BST EQU N17:1 5 NXB EQU N17:1 4 BND TON T14:13 1.0 9000 0 EOR
%   N17:1  ETAPPE_SANIT  "NR ETAPPE ACTIVE DE SANITISATION" %
% Rung: 79 %
SOR XIC T14:13/DN OTE N7:75/6 EOR
%   N7:75/6  AL43_TIME_OUT_HEAT %
% Rung: 80 %
% Alarme N°44 %
SOR EQU N17:1 10 TON T14:14 1.0 3600 0 EOR
%   N17:1  ETAPPE_SANIT  "NR ETAPPE ACTIVE DE SANITISATION" %
% Rung: 81 %
SOR XIC T14:14/DN OTE N7:75/7 EOR
%   N7:75/7  AL44_TIMEOUTFASTCOOL %
% Rung: 82 %
% Alarme N°45 %
SOR XIC B3:0/15 TON T14:15 1.0 5 0 EOR
%   B3:0/15  TSH_HX9232_B1  "Température haute TSH HX9232 B1" %
% Rung: 83 %
SOR XIC T14:15/DN OTE N7:75/8 EOR
%   N7:75/8  AL45_TSH_HX9232_B1 %

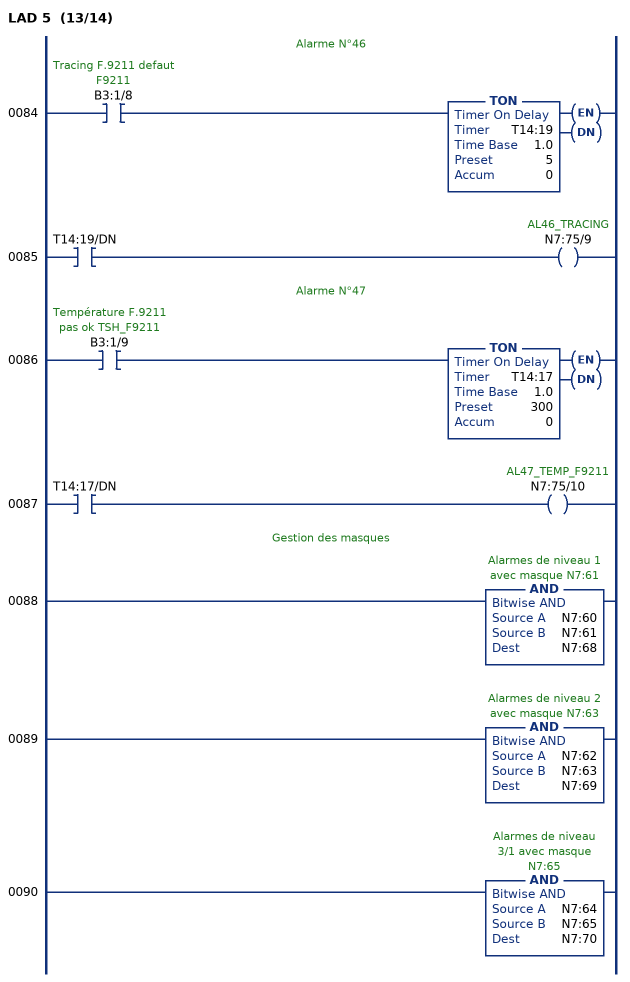
% Rung: 84 %
% Alarme N°46 %
SOR XIC B3:1/8 TON T14:19 1.0 5 0 EOR
%   B3:1/8  F9211  "Tracing F.9211 defaut" %
% Rung: 85 %
SOR XIC T14:19/DN OTE N7:75/9 EOR
%   N7:75/9  AL46_TRACING %
% Rung: 86 %
% Alarme N°47 %
SOR XIC B3:1/9 TON T14:17 1.0 300 0 EOR
%   B3:1/9  TSH_F9211  "Température F.9211 pas ok" %
% Rung: 87 %
SOR XIC T14:17/DN OTE N7:75/10 EOR
%   N7:75/10  AL47_TEMP_F9211 %
% Rung: 88 %
% Gestion des masques %
SOR AND N7:60 N7:61 N7:68 EOR
%   N7:68  "Alarmes de niveau 1 avec masque N7:61" %
% Rung: 89 %
SOR AND N7:62 N7:63 N7:69 EOR
%   N7:69  "Alarmes de niveau 2 avec masque N7:63" %
% Rung: 90 %
SOR AND N7:64 N7:65 N7:70 EOR
%   N7:70  "Alarmes de niveau 3/1 avec masque N7:65" %

